	previousNode := currentNode;
	currentNode := currentNode.Next;
	counter := counter + 1;

END_WHILE;

IF currentNode = 0 THEN
	RETURN;
END_IF

previousNode.Next := currentNode.Next;
currentNode.Next := 0;
currentNode.Destroy();
END_METHOD

END_FUNCTION_BLOCK

// ---- _Internal/Collections/CollectionNode.TcPOU
{attribute 'linkalways'} 
{attribute 'no_explicit_call' := 'This FB is a CLASS and must be accessed using methods or properties'}
{attribute 'enable_dynamic_creation'}
FUNCTION_BLOCK CollectionNode IMPLEMENTS I_CollectionNode
VAR
	collectableObject : I_Collectable;
	nextNode : I_CollectionNode;
END_VAR

PROPERTY PUBLIC Collectable : I_Collectable
GET
collectable := collectableObject;
END_GET
END_PROPERTY

METHOD PUBLIC Destroy
VAR_INPUT
END_VAR
__DELETE(THIS);
END_METHOD

METHOD FB_init : BOOL
VAR_INPUT
	bInitRetains : BOOL; // if TRUE, the retain variables are initialized (warm start / cold start)
	bInCopyCode : BOOL;  // if TRUE, the instance afterwards gets moved into the copy code (online change)
	Collectable : I_Collectable;
END_VAR
collectableObject := Collectable;
END_METHOD

PROPERTY PUBLIC Next : I_CollectionNode
GET
Next := nextNode;
END_GET
SET // PUBLIC
nextNode := Next;
END_SET
END_PROPERTY

END_FUNCTION_BLOCK

// ---- Task/Task.TcPOU
{attribute 'linkalways'} 
{attribute 'no_explicit_call' := 'This FB is a CLASS and must be accessed using methods or properties'}
{attribute 'enable_dynamic_creation'}
FUNCTION_BLOCK Task EXTENDS Instance IMPLEMENTS I_Task
VAR
	cyclicCallEvent : TaskCyclicEvent(THIS^); 
	globalInstanceMembers : GlobalInstanceMembers;
	registerInstanceToTask: RegisterInstanceToTaskCallback(Task := THIS^);
	deregisterInstanceFromTask : DeregisterInstanceFromTaskCallback(Task := THIS^);
	registerExistingInstancesToTask : RegisterInstancesToTaskVisitor(Task := THIS^);
	taskIndex : DINT;
	taskInfo : PlcTaskSystemInfo;
END_VAR

METHOD PUBLIC CyclicCall
UpdateTaskInformation();
cyclicCallEvent.Notify();
END_METHOD

METHOD PUBLIC DeregisterInstance
VAR_INPUT
	Instance : I_Instance;
END_VAR
DeregisterInstanceIfAutomaticallyCyclicCalled(Instance);
END_METHOD

METHOD PROTECTED DeregisterInstanceIfAutomaticallyCyclicCalled
VAR_INPUT
	Instance : I_Instance;
END_VAR
VAR
	cyclicInstance : I_CyclicInstance;
END_VAR
IF NOT __QUERYINTERFACE(Instance,cyclicInstance) THEN
	RETURN;
END_IF;

cyclicCallEvent.RemoveSubscriber(cyclicInstance.CyclicInstanceCallback);
END_METHOD

METHOD FB_exit : BOOL
VAR_INPUT
	bInCopyCode : BOOL; // if TRUE, the exit method is called for exiting an instance that is copied afterwards (online change).
END_VAR
globalInstanceMembers.OnInstanceAdded.RemoveSubscriber(registerInstanceToTask);
globalInstanceMembers.OnInstanceRemoved.RemoveSubscriber(deregisterInstanceFromTask);
END_METHOD

METHOD FB_init : BOOL
VAR_INPUT
	bInitRetains : BOOL; // if TRUE, the retain variables are initialized (warm start / cold start)
	bInCopyCode : BOOL;  // if TRUE, the instance afterwards gets moved into the copy code (online change)
END_VAR
globalInstanceMembers.ForEachInstance(registerExistingInstancesToTask);
globalInstanceMembers.OnInstanceAdded.AddSubscriber(RegisterInstanceToTask);
globalInstanceMembers.OnInstanceRemoved.AddSubscriber(DeregisterInstanceFromTask);
END_METHOD

PROPERTY PUBLIC Index : DINT
GET
Index := taskIndex;
END_GET
END_PROPERTY

PROPERTY Info : reference to PlcTaskSystemInfo
GET
info ref= taskInfo;
END_GET
END_PROPERTY

METHOD PUBLIC IsExecutingThis : BOOL
VAR_INPUT
END_VAR
VAR
	currentTaskIndex : DINT;
END_VAR
currentTaskIndex := GETCURTASKINDEXEX();

IF currentTaskIndex <= 0 THEN
	RETURN;
END_IF

IsExecutingThis := currentTaskIndex = taskIndex;
END_METHOD

PROPERTY PUBLIC OnCyclicCall : I_Event
GET
OnCyclicCall := cyclicCallEvent;
END_GET
END_PROPERTY

METHOD PUBLIC RegisterInstance
VAR_INPUT
	Instance : I_Instance;
END_VAR
VAR
	cyclicInstance : I_CyclicInstance;
END_VAR
RegisterInstanceIfAutomaticallyCyclicCalled(Instance);
END_METHOD

METHOD PROTECTED RegisterInstanceIfAutomaticallyCyclicCalled
VAR_INPUT
	Instance : I_Instance;
END_VAR
VAR
	cyclicInstance : I_CyclicInstance;
END_VAR
IF not __QUERYINTERFACE(Instance,cyclicInstance) THEN
	RETURN;
END_IF;

cyclicCallEvent.AddSubscriber(cyclicInstance.CyclicInstanceCallback);
END_METHOD

METHOD INTERNAL UpdateTaskInformation
taskIndex := GETCURTASKINDEXEX();
taskInfo := TwinCAT_SystemInfoVarList._TaskInfo[taskIndex];
END_METHOD

END_FUNCTION_BLOCK
